# EPICS substitutions: zfmagfldSup/zfmagfld_errors.substitutions
file $(UTILITIES)/db/error_setter.template {
    pattern {P, STREAM_PV, PV_NAME}

    {"\$(P)", "OVERLOAD", "FIELDSTRENGTH"}

}
